Omron CX-Programmer project NewProject (CX-Programmer 9.75)

# PLC ConditionalJump: CP1E N30

## Global symbols (name address type ; comment)
Condition 0.00 BOOL  ; 0.00

## Program NewProgram1 (cyclic task 0)
Local symbols
Lamp1 100.00 BOOL
Lamp2 100.01 BOOL
Sw1 0.01 BOOL
Sw2 0.02 BOOL

### Section Section1

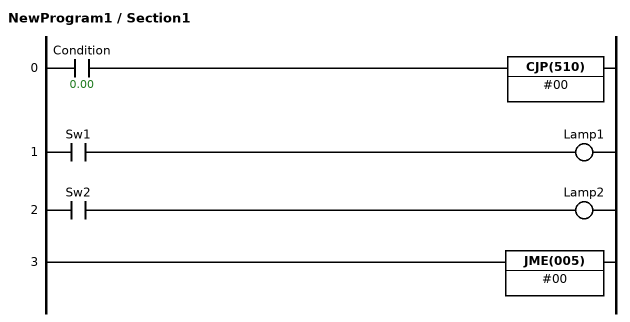
; rung 0
LD Condition  ; 0.00
CJP(510) #00
; rung 1
LD Sw1
OUT Lamp1
; rung 2
LD Sw2
OUT Lamp2
; rung 3
JME(005) #00

### Section END
; rung 0
END(001)